FUNCTION_BLOCK Model (* Composite Function Block Type *)
  (* Standard: 61499-2 *)
  (* Version 0.0, 7/13/2016, Andrei, nxtControl GmbH, template *)
  PACKAGE Main;
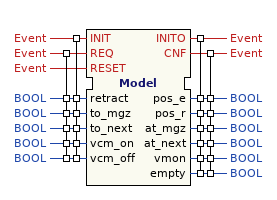
  EVENT_INPUT
    INIT WITH retract, to_mgz, to_next, vcm_off, vcm_on; (* Initialization Request *)
    REQ WITH retract, to_mgz, to_next, vcm_off, vcm_on; (* Normal Execution Request *)
    RESET;
  END_EVENT
  EVENT_OUTPUT
    INITO WITH pos_e, pos_r, at_mgz, at_next, vmon, empty; (* Initialization Confirm *)
    CNF WITH pos_e, pos_r, at_mgz, at_next, vmon, empty; (* Execution Confirmation *)
  END_EVENT
  VAR_INPUT
    retract : BOOL; (* Input event qualifier *)
    to_mgz : BOOL;
    to_next : BOOL;
    vcm_on : BOOL;
    vcm_off : BOOL;
  END_VAR
  VAR_OUTPUT
    pos_e : BOOL; (* Output event qualifier *)
    pos_r : BOOL;
    at_mgz : BOOL;
    at_next : BOOL;
    vmon : BOOL;
    empty : BOOL;
  END_VAR
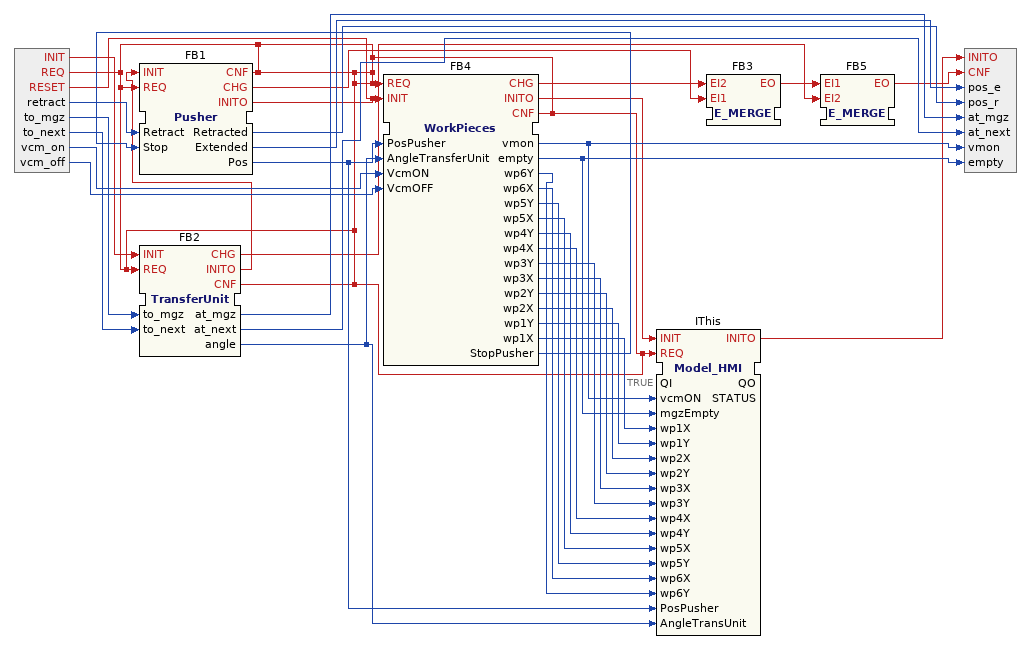
  FBS
    FB3 : E_MERGE;
    FB5 : E_MERGE;
    FB2 : TransferUnit;
    FB4 : WorkPieces;
    IThis : Model_HMI(QI := TRUE);
    FB1 : Pusher;
  END_FBS
  EVENT_CONNECTIONS
    FB1.CNF TO FB4.REQ;
    FB4.CHG TO FB3.EI2;
    FB1.CHG TO FB3.EI1;
    FB3.EO TO FB5.EI1;
    FB2.CHG TO FB5.EI2;
    FB2.INITO TO FB1.INIT;
    INIT TO FB2.INIT;
    REQ TO FB1.REQ;
    REQ TO FB2.REQ;
    FB1.INITO TO FB4.INIT;
    FB2.CNF TO FB4.REQ;
    FB5.EO TO CNF;
    IThis.INITO TO INITO;
    FB4.INITO TO IThis.INIT;
    FB4.CNF TO IThis.REQ;
    FB2.CNF TO IThis.REQ;
    FB1.CNF TO IThis.REQ;
    REQ TO FB4.REQ;
    FB4.CNF TO FB1.REQ;
    FB4.CNF TO FB2.REQ;
    RESET TO FB4.INIT;
  END_CONNECTIONS
  DATA_CONNECTIONS
    to_mgz TO FB2.to_mgz;
    to_next TO FB2.to_next;
    FB2.at_mgz TO at_mgz;
    FB2.at_next TO at_next;
    FB1.Retracted TO pos_r;
    FB1.Extended TO pos_e;
    retract TO FB1.Retract;
    FB1.Pos TO FB4.PosPusher;
    FB2.angle TO FB4.AngleTransferUnit;
    FB4.vmon TO vmon;
    FB4.empty TO empty;
    FB2.angle TO IThis.AngleTransUnit;
    FB1.Pos TO IThis.PosPusher;
    FB4.wp6Y TO IThis.wp6Y;
    FB4.wp6X TO IThis.wp6X;
    FB4.wp5Y TO IThis.wp5Y;
    FB4.wp5X TO IThis.wp5X;
    FB4.wp4Y TO IThis.wp4Y;
    FB4.wp4X TO IThis.wp4X;
    FB4.wp3Y TO IThis.wp3Y;
    FB4.wp3X TO IThis.wp3X;
    FB4.wp2Y TO IThis.wp2Y;
    FB4.wp2X TO IThis.wp2X;
    FB4.wp1Y TO IThis.wp1Y;
    FB4.wp1X TO IThis.wp1X;
    FB4.StopPusher TO FB1.Stop;
    FB4.vmon TO IThis.vcmON;
    FB4.empty TO IThis.mgzEmpty;
    vcm_on TO FB4.VcmON;
    vcm_off TO FB4.VcmOFF;
  END_CONNECTIONS
END_FUNCTION_BLOCK
